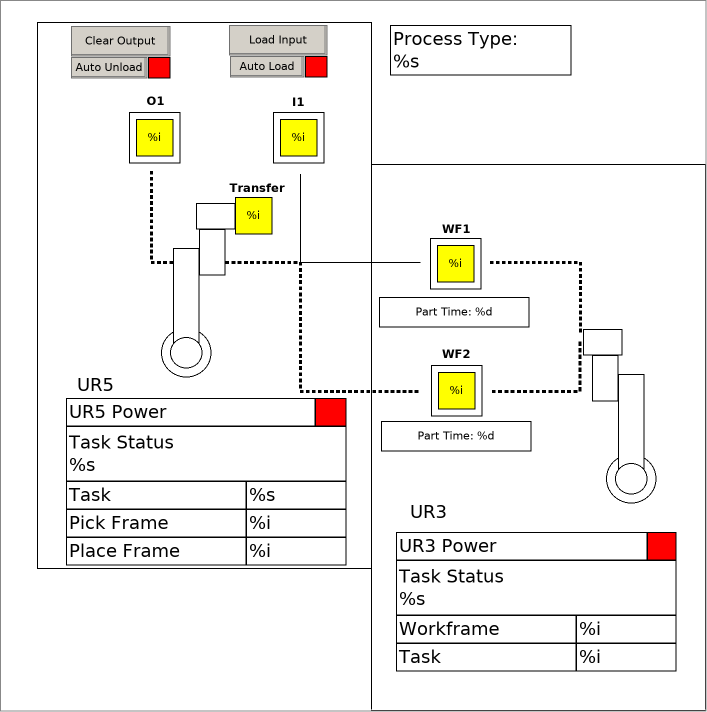
VISUALIZATION Process  // 707x712
    Rectangle (235,197 37x37)
    Line (371,164) (705,164)
    Line (371,710) (705,710)
    Line (705,164) (705,709)
    Line (371,164) (371,709)
    Rectangle (430,238 51x51), colour toggle: Global.arrWorkFixtures[1].bReserved
    Rectangle (431,365 51x51), colour toggle: Global.arrWorkFixtures[2].bReserved
    Rectangle (437,245 37x37), "%i", text variable: Global.arrWorkFixtures[1].stPart.nPartNumber, colour toggle: Global.arrWorkFixtures[1].stPart.bComplete, invisible if: NOT Global.arrWorkFixtures[1].stPart.bExists
    Rectangle (438,372 37x37), "%i", text variable: Global.arrWorkFixtures[2].stPart.nPartNumber, colour toggle: Global.arrWorkFixtures[2].stPart.bComplete, invisible if: NOT Global.arrWorkFixtures[2].stPart.bExists
    Rectangle (379,297 150x30), "Part Time: %d", text variable: Global.arrWorkFixtures[1].stPart.ntTimeInWorkfixture
    Rectangle (381,421 150x30), "Part Time: %d", text variable: Global.arrWorkFixtures[2].stPart.ntTimeInWorkfixture
    Line (37,22) (371,22)
    Line (37,568) (371,568)
    Line (371,22) (371,567)
    Line (37,23) (37,568)
    Label (67,370 57x30), "UR5"
    Rectangle (273,112 51x51), colour toggle: Global.arrInputFixtures[1].bReserved
    Rectangle (280,119 37x37), "%i", text variable: Global.arrInputFixtures[1].stPart.nPartNumber, colour toggle: Global.arrInputFixtures[1].stPart.bComplete, invisible if: NOT Global.arrInputFixtures[1].stPart.bExists
    Rectangle (129,112 51x51), colour toggle: Global.arrOutputFixtures[1].bReserved
    Rectangle (136,119 37x37), "%i", text variable: Global.arrOutputFixtures[1].stPart.nPartNumber, colour toggle: Global.arrOutputFixtures[1].stPart.bComplete, invisible if: NOT Global.arrOutputFixtures[1].stPart.bExists
    Button (229,25 98x30), "Load Input"
        OnMouseClick: execute { P_InputOutputHandling.bAddParts := TRUE; }
    Button (71,26 99x30), "Clear Output"
        OnMouseClick: execute { P_InputOutputHandling.bRemoveParts := true; }
    Line (300,262) (420,262), colour toggle: P_TaskHandling.stUR5TaskStatus.bInTask AND (P_TaskHandling.nUR5TargetPickFrame = Global.arrWorkFixtures[1].nWorkframe OR P_TaskHandling.nUR5TargetPlaceFrame = Global.arrWorkFixtures[1].nWorkframe)
    Line (300,174) (300,262), colour toggle: P_TaskHandling.nUR5TargetTask = 1
    Polyline (151,171) (151,262) (300,262), colour toggle: P_TaskHandling.nUR5TargetTask = 2
    Polyline (300,262) (300,391) (421,391), colour toggle: P_TaskHandling.stUR5TaskStatus.bInTask AND (P_TaskHandling.nUR5TargetPickFrame = Global.arrWorkFixtures[2].nWorkframe OR P_TaskHandling.nUR5TargetPlaceFrame = Global.arrWorkFixtures[2].nWorkframe)
    Rectangle (235,197 37x37), "%i", text variable: Global.stPartInTransit.nPartNumber, colour toggle: Global.stPartInTransit.bComplete, invisible if: NOT Global.stPartInTransit.bExists
    Polyline (490,262) (580,262) (580,335), colour toggle: P_TaskHandling.nUR3TargetWorkFixtureIndex = 1
    Polyline (492,391) (580,391) (580,339), colour toggle: P_TaskHandling.nUR3TargetWorkFixtureIndex = 2
    Rectangle (396,532 251x28), "UR3 Power"
    Rectangle (647,532 29x28), colour toggle: Global_Safety.UR3RedIND
    Rectangle (396,560 280x55), "Task Status %s", text variable: P_TaskHandling.stUR3TaskStatus.sRobotStatus
    Rectangle (396,615 180x28), "Workframe"
    Rectangle (576,615 100x28), "%i", text variable: P_TaskHandling.nUR3TargetWorkframe
    Rectangle (396,643 180x28), "Task"
    Rectangle (576,643 100x28), "%i", text variable: P_TaskHandling.nUR3TargetTask
    Rectangle (66,398 249x28), "UR5 Power"
    Rectangle (315,398 31x28), colour toggle: Global_Safety.UR5RedIND
    Rectangle (66,426 280x55), "Task Status %s", text variable: P_TaskHandling.stUR5TaskStatus.sRobotStatus
    Rectangle (66,481 180x28), "Task"
    Rectangle (246,481 100x28), "%s", text variable: P_TaskHandling.sUR5TargetTask
    Rectangle (66,509 180x28), "Pick Frame"
    Rectangle (246,509 100x28), "%i", text variable: P_TaskHandling.nUR5TargetPickFrame
    Label (400,497 57x30), "UR3"
    Rectangle (66,537 180x28), "Place Frame"
    Rectangle (246,537 100x28), "%i", text variable: P_TaskHandling.nUR5TargetPlaceFrame
    Group (161,203 74x174)
        Ellipse (0,125 50x49), colour toggle: Global_Safety.UR5RedIND
        Group (9,0 65x165)
            Rectangle (3,45 26x103)
            Rectangle (26,0 39x26)
            Ellipse (0,134 32x31)
            Rectangle (29,26 26x46)
    Group (583,329 73x174)
        Ellipse (23,125 50x49), colour toggle: Global_Safety.UR3RedIND
        Rectangle (35,45 26x103)
        Rectangle (0,0 39x26)
        Ellipse (32,134 32x31)
        Rectangle (9,26 26x46)
    Label (428,339 57x30), "WF2"
    Label (428,214 57x30), "WF1"
    Label (225,173 64x30), "Transfer"
    Label (270,87 57x30), "I1"
    Label (127,86 57x30), "O1"
    Rectangle (390,25 181x50), "Process Type: %s", text variable: P_InputOutputHandling.sProcessType
    Button (71,57 76x21), "Auto Unload"
        OnMouseClick: toggle P_InputOutputHandling.bAutoUnload
    Button (230,56 74x21), "Auto Load"
        OnMouseClick: toggle P_InputOutputHandling.bAutoLoad
    Rectangle (148,57 22x21), colour toggle: P_InputOutputHandling.bAutoUnload
    Rectangle (305,56 22x21), colour toggle: P_InputOutputHandling.bAutoLoad
END_VISUALIZATION

(* stored: Version 1.1.0.1, ProductVersion 3.1.4020.12
   Visu Process: Id {2e1481f5-8124-4d07-a6b7-91970834a754} *)
